ABB RAPID module: 002B12D6

MODULE MainModule

    CONST jointtarget jtHome:=[[0,0,0,0,0,0],[9E+09,9E+09,9E+09,9E+09,9E+09,9E+09]];

    CONST robtarget pStart := [[0,0,500],[0,0,1,0],[0,0,0,0],[9E+09,9E+09,9E+09,9E+09,9E+09,9E+09]];
    CONST robtarget pStart_1 := [[0,400,500],[0,0,1,0],[0,0,0,0],[9E+09,9E+09,9E+09,9E+09,9E+09,9E+09]];

    !Shape_0

    PROC main()

        !MoveAbsJ jtHome,v1000,fine,tool0;

        MoveJ pStart,v1000,fine,Weldgun\WObj:=Level_0;
        !MoveJ pStart_1,v1000,fine,Weldgun\WObj:=Level_0;
        Shape_1_Move_0;

    ENDPROC


ENDMODULE
